(* PLC project v0.6.04_CycleSemiAuto.project, CODESYS CODESYS V3.5 SP19 Patch 1 *)
(* stored: creationDateTime 2026-08-17T05:53:47.257609, modificationDateTime 2026-08-17T05:53:47.257609 *)

(* ═══════════════════════════════════════════════════════════════ 🔧 ST_SyncCfg — Configuration de la synchronisation M1/M2 ═══════════════════════════════════════════════════════════════ *)
TYPE ST_SyncCfg : STRUCT
  CfgSyncTolerance_M : REAL := 0.8;  (* 📐 Tolérance max d'écart (m) — Dégradation Palier 1 dès 0.8m *)
  Initialized : BOOL := FALSE;  (* 🚦 flag restauration boot, ex-CfgInitialized renommé pour cohérence avec ST_WinchCfg *)
END_STRUCT;
END_TYPE
